SYSTEM CONVEYORS (* System Configuration *)
  (* Standard: 61499-1 *)
  (* Version 0.4, 2009-03-05, JHC, Holobloc Inc., Deleted Application. *)
  (* Version 0.3, 2003-12-05, JHC, Rockwell Automation, Renamed from NEWSYSTEM. *)
  (* Version 0.2, 2002-11-05, JHC, Rockwell Automation, Fixed missing (empty) FBD in Application. *)
  (* Version 0.1, 2002-01-17, JHC, Rockwell Automation, Minor cleanup *)
  (* Version 0.0, 2000-05-27, JHC, Rockwell Automation *)
  DEVICE VIEW : FRAME_DEVICE(BOUNDS := [500,30,520,500])
    RESOURCE VIEW_Resource : VIEW_PANEL(DIA := 50, SIZE := [10,10])
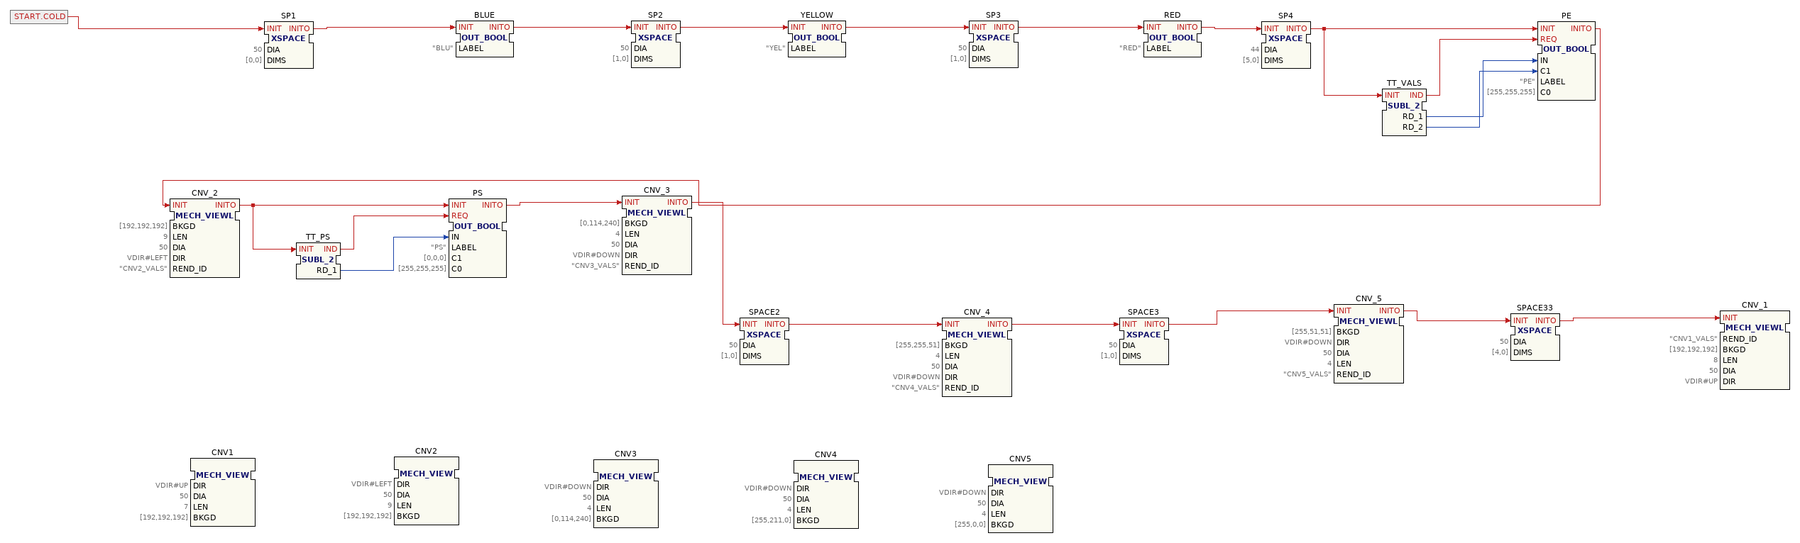
      FBS
        CNV1 : MECH_VIEW(DIR := VDIR#UP, DIA := 50, LEN := 7, BKGD := [192,192,192]);
        CNV2 : MECH_VIEW(DIR := VDIR#LEFT, DIA := 50, LEN := 9, BKGD := [192,192,192]);
        CNV3 : MECH_VIEW(DIR := VDIR#DOWN, DIA := 50, LEN := 4, BKGD := [0,114,240]);
        CNV4 : MECH_VIEW(DIR := VDIR#DOWN, DIA := 50, LEN := 4, BKGD := [255,211,0]);
        CNV5 : MECH_VIEW(DIR := VDIR#DOWN, DIA := 50, LEN := 4, BKGD := [255,0,0]);
        SPACE2 : XSPACE(DIA := 50, DIMS := [1,0]);
        SPACE3 : XSPACE(DIA := 50, DIMS := [1,0]);
        BLUE : OUT_BOOL(LABEL := "BLU");
        YELLOW : OUT_BOOL(LABEL := "YEL");
        RED : OUT_BOOL(LABEL := "RED");
        SP1 : XSPACE(DIA := 50, DIMS := [0,0]);
        SP2 : XSPACE(DIA := 50, DIMS := [1,0]);
        SP3 : XSPACE(DIA := 50, DIMS := [1,0]);
        SP4 : XSPACE(DIA := 44, DIMS := [5,0]);
        SPACE33 : XSPACE(DIA := 50, DIMS := [4,0]);
        PS : OUT_BOOL(LABEL := "PS", C1 := [0,0,0], C0 := [255,255,255]);
        PE : OUT_BOOL(LABEL := "PE", C0 := [255,255,255]);
        CNV_2 : MECH_VIEWL(BKGD := [192,192,192], LEN := 9, DIA := 50, DIR := VDIR#LEFT, REND_ID := "CNV2_VALS");
        CNV_3 : MECH_VIEWL(BKGD := [0,114,240], LEN := 4, DIA := 50, DIR := VDIR#DOWN, REND_ID := "CNV3_VALS");
        CNV_4 : MECH_VIEWL(BKGD := [255,255,51], LEN := 4, DIA := 50, DIR := VDIR#DOWN, REND_ID := "CNV4_VALS");
        CNV_5 : MECH_VIEWL(BKGD := [255,51,51], DIR := VDIR#DOWN, DIA := 50, LEN := 4, REND_ID := "CNV5_VALS");
        TT_VALS : SUBL_2;
        TT_PS : SUBL_2;
        CNV_1 : MECH_VIEWL(REND_ID := "CNV1_VALS", BKGD := [192,192,192], LEN := 8, DIA := 50, DIR := VDIR#UP);
      END_FBS
      EVENT_CONNECTIONS
        START.COLD TO SP1.INIT;
        SP1.INITO TO BLUE.INIT;
        BLUE.INITO TO SP2.INIT;
        SP2.INITO TO YELLOW.INIT;
        YELLOW.INITO TO SP3.INIT;
        SP3.INITO TO RED.INIT;
        RED.INITO TO SP4.INIT;
        SP4.INITO TO PE.INIT;
        PE.INITO TO CNV_2.INIT;
        CNV_2.INITO TO PS.INIT;
        PS.INITO TO CNV_3.INIT;
        CNV_3.INITO TO SPACE2.INIT;
        SPACE2.INITO TO CNV_4.INIT;
        CNV_4.INITO TO SPACE3.INIT;
        SPACE3.INITO TO CNV_5.INIT;
        CNV_5.INITO TO SPACE33.INIT;
        SP4.INITO TO TT_VALS.INIT;
        TT_VALS.IND TO PE.REQ;
        CNV_2.INITO TO TT_PS.INIT;
        TT_PS.IND TO PS.REQ;
        SPACE33.INITO TO CNV_1.INIT;
      END_CONNECTIONS
      DATA_CONNECTIONS
        TT_VALS.RD_1 TO PE.IN;
        TT_VALS.RD_2 TO PE.C1;
        TT_PS.RD_1 TO PS.IN;
      END_CONNECTIONS
    END_RESOURCE
  END_DEVICE
  DEVICE HMI : FRAME_DEVICE(BOUNDS := [1000,30,500,500])
    RESOURCE HMI_RESOURCE : VIEW_PANEL(DIA := 50, SIZE := [10,10])
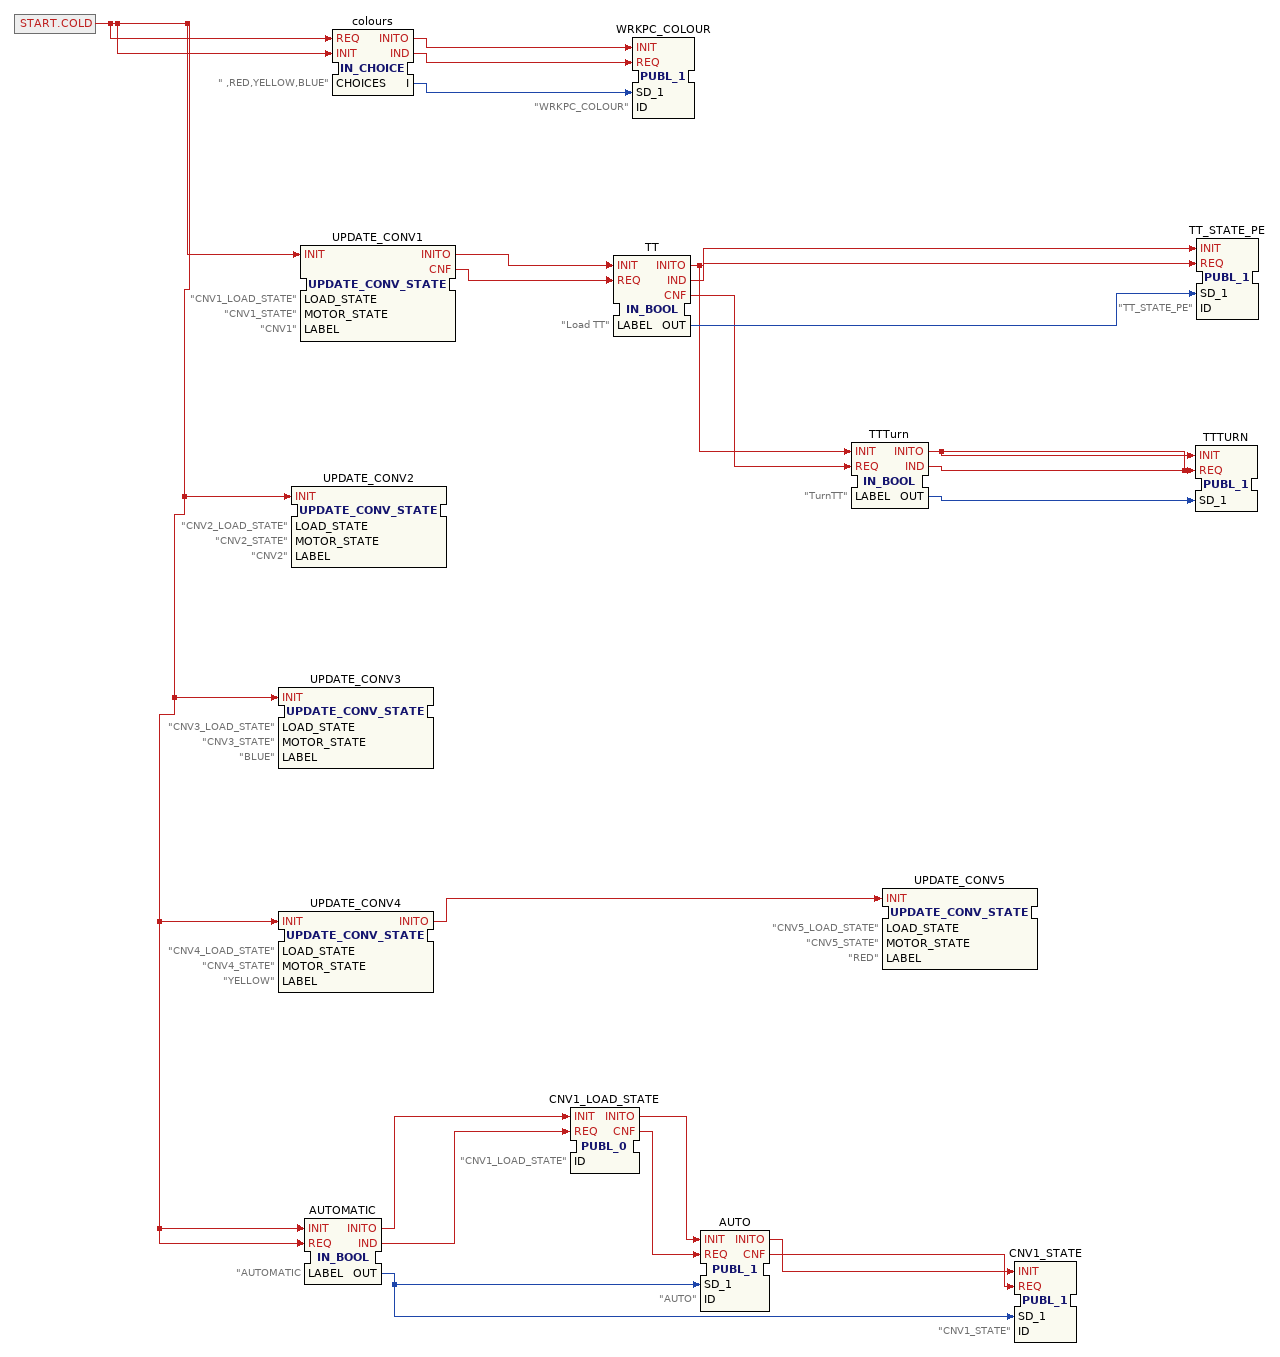
      FBS
        colours : IN_CHOICE(CHOICES := " ,RED,YELLOW,BLUE");
        WRKPC_COLOUR : PUBL_1(ID := "WRKPC_COLOUR");
        TT_STATE_PE : PUBL_1(ID := "TT_STATE_PE");
        TT : IN_BOOL(LABEL := "Load TT");
        TTTurn : IN_BOOL(LABEL := "TurnTT");
        TTTURN : PUBL_1;
        UPDATE_CONV1 : UPDATE_CONV_STATE(LOAD_STATE := "CNV1_LOAD_STATE", MOTOR_STATE := "CNV1_STATE", LABEL := "CNV1");
        UPDATE_CONV2 : UPDATE_CONV_STATE(LOAD_STATE := "CNV2_LOAD_STATE", MOTOR_STATE := "CNV2_STATE", LABEL := "CNV2");
        UPDATE_CONV3 : UPDATE_CONV_STATE(LOAD_STATE := "CNV3_LOAD_STATE", MOTOR_STATE := "CNV3_STATE", LABEL := "BLUE");
        UPDATE_CONV4 : UPDATE_CONV_STATE(LOAD_STATE := "CNV4_LOAD_STATE", MOTOR_STATE := "CNV4_STATE", LABEL := "YELLOW");
        UPDATE_CONV5 : UPDATE_CONV_STATE(LOAD_STATE := "CNV5_LOAD_STATE", MOTOR_STATE := "CNV5_STATE", LABEL := "RED");
        AUTOMATIC : IN_BOOL(LABEL := "AUTOMATIC);
        CNV1_STATE : PUBL_1(ID := "CNV1_STATE");
        CNV1_LOAD_STATE : PUBL_0(ID := "CNV1_LOAD_STATE");
        AUTO : PUBL_1(ID := "AUTO");
      END_FBS
      EVENT_CONNECTIONS
        START.COLD TO colours.REQ;
        START.COLD TO colours.INIT;
        colours.INITO TO WRKPC_COLOUR.INIT;
        colours.IND TO WRKPC_COLOUR.REQ;
        TT.INITO TO TT_STATE_PE.INIT;
        TT.IND TO TT_STATE_PE.REQ;
        TT.INITO TO TTTurn.INIT;
        TT.CNF TO TTTurn.REQ;
        TTTurn.INITO TO TTTURN.INIT;
        TTTurn.IND TO TTTURN.REQ;
        TTTurn.INITO TO TTTURN.REQ;
        START.COLD TO UPDATE_CONV1.INIT;
        UPDATE_CONV1.INITO TO TT.INIT;
        UPDATE_CONV1.CNF TO TT.REQ;
        START.COLD TO UPDATE_CONV2.INIT;
        START.COLD TO UPDATE_CONV3.INIT;
        START.COLD TO UPDATE_CONV4.INIT;
        UPDATE_CONV4.INITO TO UPDATE_CONV5.INIT;
        START.COLD TO AUTOMATIC.INIT;
        START.COLD TO AUTOMATIC.REQ;
        AUTOMATIC.INITO TO CNV1_LOAD_STATE.INIT;
        AUTOMATIC.IND TO CNV1_LOAD_STATE.REQ;
        CNV1_LOAD_STATE.INITO TO AUTO.INIT;
        CNV1_LOAD_STATE.CNF TO AUTO.REQ;
        AUTO.INITO TO CNV1_STATE.INIT;
        AUTO.CNF TO CNV1_STATE.REQ;
      END_CONNECTIONS
      DATA_CONNECTIONS
        colours.I TO WRKPC_COLOUR.SD_1;
        TT.OUT TO TT_STATE_PE.SD_1;
        TTTurn.OUT TO TTTURN.SD_1;
        AUTOMATIC.OUT TO CNV1_STATE.SD_1;
        AUTOMATIC.OUT TO AUTO.SD_1;
      END_CONNECTIONS
    END_RESOURCE
  END_DEVICE
  DEVICE MODEL : FRAME_DEVICE(BOUNDS := [500,570,500,500])
    RESOURCE CONV1_MODEL : VIEW_PANEL(DIA := 50, SIZE := [1,1])
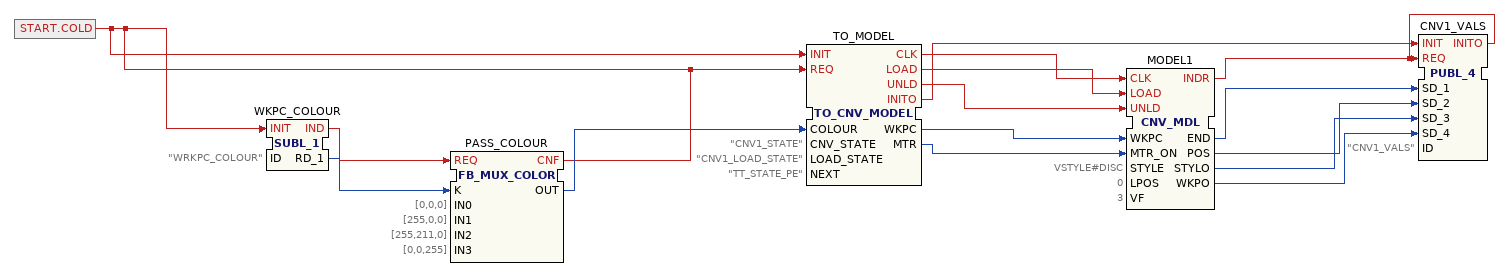
      FBS
        MODEL1 : CNV_MDL(STYLE := VSTYLE#DISC, LPOS := 0, VF := 3);
        TO_MODEL : TO_CNV_MODEL(CNV_STATE := "CNV1_STATE", LOAD_STATE := "CNV1_LOAD_STATE", NEXT := "TT_STATE_PE");
        CNV1_VALS : PUBL_4(ID := "CNV1_VALS");
        WKPC_COLOUR : SUBL_1(ID := "WRKPC_COLOUR");
        PASS_COLOUR : FB_MUX_COLOR(IN0 := [0,0,0], IN1 := [255,0,0], IN2 := [255,211,0], IN3 := [0,0,255]);
      END_FBS
      EVENT_CONNECTIONS
        START.COLD TO TO_MODEL.INIT;
        TO_MODEL.CLK TO MODEL1.CLK;
        START.COLD TO TO_MODEL.REQ;
        TO_MODEL.LOAD TO MODEL1.LOAD;
        TO_MODEL.UNLD TO MODEL1.UNLD;
        TO_MODEL.INITO TO CNV1_VALS.INIT;
        MODEL1.INDR TO CNV1_VALS.REQ;
        CNV1_VALS.INITO TO CNV1_VALS.REQ;
        START.COLD TO WKPC_COLOUR.INIT;
        WKPC_COLOUR.IND TO PASS_COLOUR.REQ;
        PASS_COLOUR.CNF TO TO_MODEL.REQ;
      END_CONNECTIONS
      DATA_CONNECTIONS
        TO_MODEL.WKPC TO MODEL1.WKPC;
        TO_MODEL.MTR TO MODEL1.MTR_ON;
        MODEL1.END TO CNV1_VALS.SD_1;
        MODEL1.POS TO CNV1_VALS.SD_2;
        MODEL1.STYLO TO CNV1_VALS.SD_3;
        MODEL1.WKPO TO CNV1_VALS.SD_4;
        WKPC_COLOUR.RD_1 TO PASS_COLOUR.K;
        PASS_COLOUR.OUT TO TO_MODEL.COLOUR;
      END_CONNECTIONS
    END_RESOURCE
    RESOURCE TT_MODEL : VIEW_PANEL(DIA := 50, SIZE := [1,1])
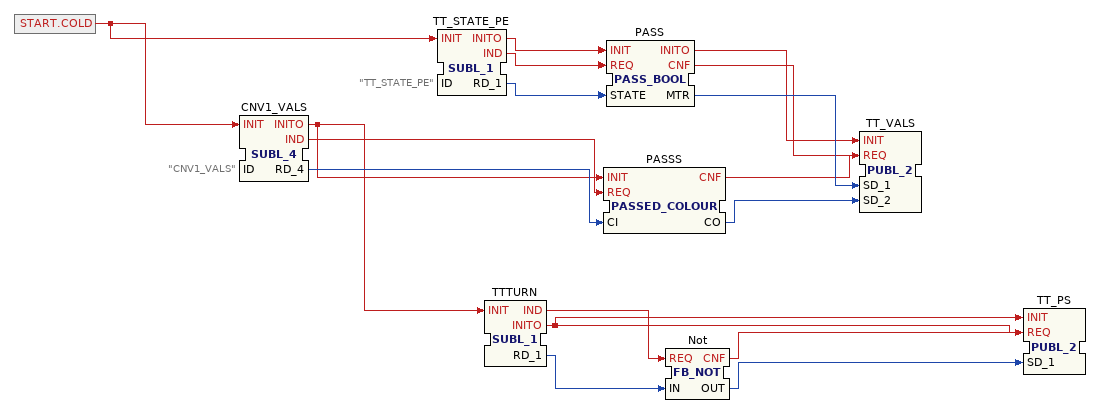
      FBS
        TT_STATE_PE : SUBL_1(ID := "TT_STATE_PE");
        TT_PS : PUBL_2;
        TTTURN : SUBL_1;
        Not : FB_NOT;
        CNV1_VALS : SUBL_4(ID := "CNV1_VALS");
        PASS : PASS_BOOL;
        PASSS : PASSED_COLOUR;
        TT_VALS : PUBL_2;
      END_FBS
      EVENT_CONNECTIONS
        START.COLD TO TT_STATE_PE.INIT;
        TTTURN.IND TO Not.REQ;
        TTTURN.INITO TO TT_PS.INIT;
        Not.CNF TO TT_PS.REQ;
        TTTURN.INITO TO TT_PS.REQ;
        START.COLD TO CNV1_VALS.INIT;
        CNV1_VALS.INITO TO TTTURN.INIT;
        TT_STATE_PE.INITO TO PASS.INIT;
        TT_STATE_PE.IND TO PASS.REQ;
        CNV1_VALS.INITO TO PASSS.INIT;
        CNV1_VALS.IND TO PASSS.REQ;
        PASS.INITO TO TT_VALS.INIT;
        PASS.CNF TO TT_VALS.REQ;
        PASSS.CNF TO TT_VALS.REQ;
      END_CONNECTIONS
      DATA_CONNECTIONS
        Not.OUT TO TT_PS.SD_1;
        TTTURN.RD_1 TO Not.IN;
        TT_STATE_PE.RD_1 TO PASS.STATE;
        CNV1_VALS.RD_4 TO PASSS.CI;
        PASS.MTR TO TT_VALS.SD_1;
        PASSS.CO TO TT_VALS.SD_2;
      END_CONNECTIONS
    END_RESOURCE
    RESOURCE CONV2_MODEL : VIEW_PANEL(DIA := 50, SIZE := [1,1])
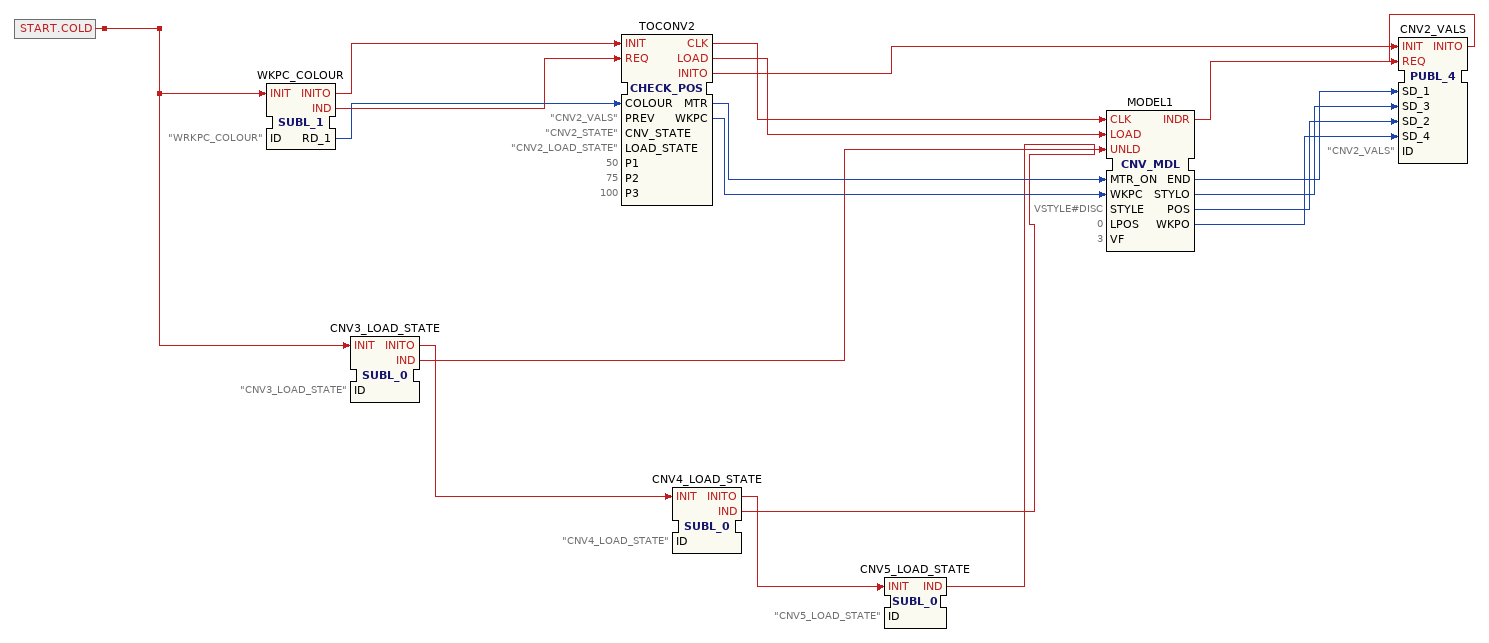
      FBS
        MODEL1 : CNV_MDL(STYLE := VSTYLE#DISC, LPOS := 0, VF := 3);
        TOCONV2 : CHECK_POS(PREV := "CNV2_VALS", CNV_STATE := "CNV2_STATE", LOAD_STATE := "CNV2_LOAD_STATE", P1 := 50, P2 := 75, P3 := 100);
        CNV3_LOAD_STATE : SUBL_0(ID := "CNV3_LOAD_STATE");
        CNV4_LOAD_STATE : SUBL_0(ID := "CNV4_LOAD_STATE");
        CNV5_LOAD_STATE : SUBL_0(ID := "CNV5_LOAD_STATE");
        CNV2_VALS : PUBL_4(ID := "CNV2_VALS");
        WKPC_COLOUR : SUBL_1(ID := "WRKPC_COLOUR");
      END_FBS
      EVENT_CONNECTIONS
        TOCONV2.CLK TO MODEL1.CLK;
        TOCONV2.LOAD TO MODEL1.LOAD;
        CNV3_LOAD_STATE.INITO TO CNV4_LOAD_STATE.INIT;
        CNV4_LOAD_STATE.INITO TO CNV5_LOAD_STATE.INIT;
        TOCONV2.INITO TO CNV2_VALS.INIT;
        MODEL1.INDR TO CNV2_VALS.REQ;
        CNV2_VALS.INITO TO CNV2_VALS.REQ;
        START.COLD TO WKPC_COLOUR.INIT;
        WKPC_COLOUR.INITO TO TOCONV2.INIT;
        WKPC_COLOUR.IND TO TOCONV2.REQ;
        START.COLD TO CNV3_LOAD_STATE.INIT;
        CNV3_LOAD_STATE.IND TO MODEL1.UNLD;
        CNV4_LOAD_STATE.IND TO MODEL1.UNLD;
        CNV5_LOAD_STATE.IND TO MODEL1.UNLD;
      END_CONNECTIONS
      DATA_CONNECTIONS
        TOCONV2.MTR TO MODEL1.MTR_ON;
        TOCONV2.WKPC TO MODEL1.WKPC;
        MODEL1.END TO CNV2_VALS.SD_1;
        MODEL1.STYLO TO CNV2_VALS.SD_3;
        MODEL1.POS TO CNV2_VALS.SD_2;
        MODEL1.WKPO TO CNV2_VALS.SD_4;
        WKPC_COLOUR.RD_1 TO TOCONV2.COLOUR;
      END_CONNECTIONS
    END_RESOURCE
    RESOURCE CONV3_MODEL : VIEW_PANEL(DIA := 50, SIZE := [1,1])
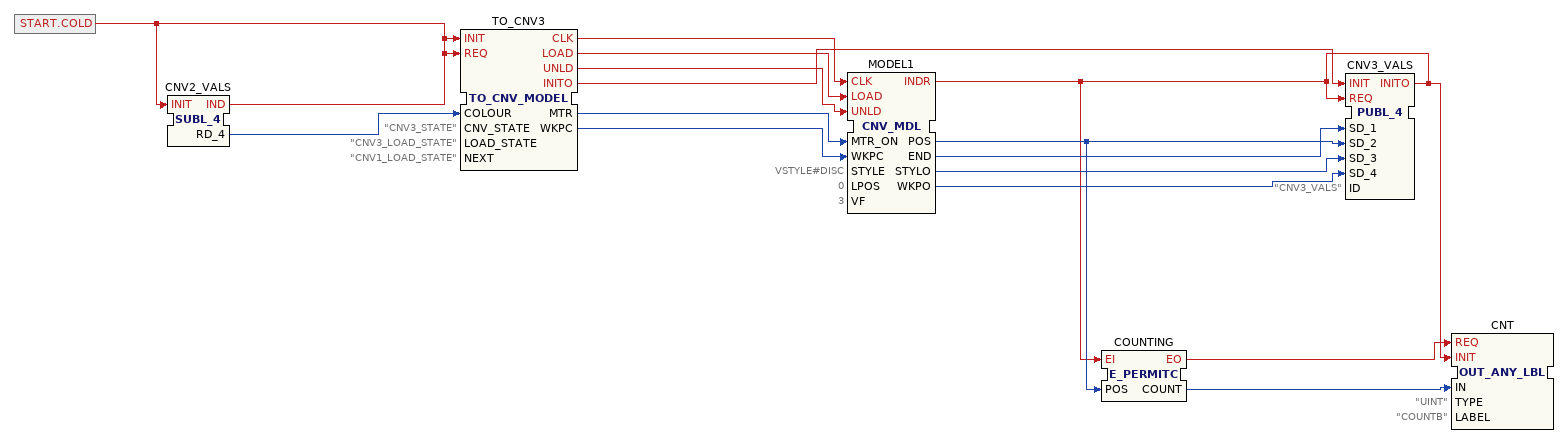
      FBS
        MODEL1 : CNV_MDL(STYLE := VSTYLE#DISC, LPOS := 0, VF := 3);
        TO_CNV3 : TO_CNV_MODEL(CNV_STATE := "CNV3_STATE", LOAD_STATE := "CNV3_LOAD_STATE", NEXT := "CNV1_LOAD_STATE");
        COUNTING : E_PERMITC;
        CNT : OUT_ANY_LBL(TYPE := "UINT", LABEL := "COUNTB");
        CNV3_VALS : PUBL_4(ID := "CNV3_VALS");
        CNV2_VALS : SUBL_4;
      END_FBS
      EVENT_CONNECTIONS
        START.COLD TO TO_CNV3.INIT;
        START.COLD TO TO_CNV3.REQ;
        TO_CNV3.CLK TO MODEL1.CLK;
        TO_CNV3.LOAD TO MODEL1.LOAD;
        TO_CNV3.UNLD TO MODEL1.UNLD;
        MODEL1.INDR TO COUNTING.EI;
        COUNTING.EO TO CNT.REQ;
        TO_CNV3.INITO TO CNV3_VALS.INIT;
        MODEL1.INDR TO CNV3_VALS.REQ;
        CNV3_VALS.INITO TO CNV3_VALS.REQ;
        CNV3_VALS.INITO TO CNT.INIT;
        START.COLD TO CNV2_VALS.INIT;
        CNV2_VALS.IND TO TO_CNV3.REQ;
      END_CONNECTIONS
      DATA_CONNECTIONS
        TO_CNV3.MTR TO MODEL1.MTR_ON;
        TO_CNV3.WKPC TO MODEL1.WKPC;
        MODEL1.POS TO COUNTING.POS;
        COUNTING.COUNT TO CNT.IN;
        MODEL1.END TO CNV3_VALS.SD_1;
        MODEL1.POS TO CNV3_VALS.SD_2;
        MODEL1.STYLO TO CNV3_VALS.SD_3;
        MODEL1.WKPO TO CNV3_VALS.SD_4;
        CNV2_VALS.RD_4 TO TO_CNV3.COLOUR;
      END_CONNECTIONS
    END_RESOURCE
    RESOURCE CONV4_MODEL : VIEW_PANEL(DIA := 50, SIZE := [1,1])
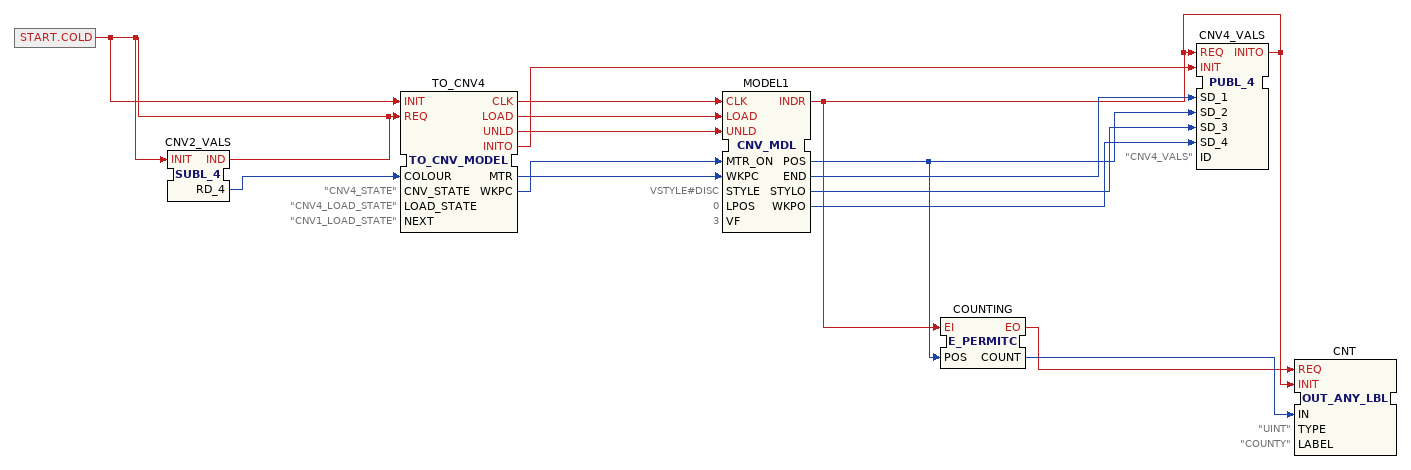
      FBS
        MODEL1 : CNV_MDL(STYLE := VSTYLE#DISC, LPOS := 0, VF := 3);
        TO_CNV4 : TO_CNV_MODEL(CNV_STATE := "CNV4_STATE", LOAD_STATE := "CNV4_LOAD_STATE", NEXT := "CNV1_LOAD_STATE");
        COUNTING : E_PERMITC;
        CNT : OUT_ANY_LBL(TYPE := "UINT", LABEL := "COUNTY");
        CNV4_VALS : PUBL_4(ID := "CNV4_VALS");
        CNV2_VALS : SUBL_4;
      END_FBS
      EVENT_CONNECTIONS
        START.COLD TO TO_CNV4.INIT;
        TO_CNV4.CLK TO MODEL1.CLK;
        TO_CNV4.LOAD TO MODEL1.LOAD;
        TO_CNV4.UNLD TO MODEL1.UNLD;
        START.COLD TO TO_CNV4.REQ;
        MODEL1.INDR TO COUNTING.EI;
        COUNTING.EO TO CNT.REQ;
        CNV4_VALS.INITO TO CNV4_VALS.REQ;
        TO_CNV4.INITO TO CNV4_VALS.INIT;
        MODEL1.INDR TO CNV4_VALS.REQ;
        CNV4_VALS.INITO TO CNT.INIT;
        START.COLD TO CNV2_VALS.INIT;
        CNV2_VALS.IND TO TO_CNV4.REQ;
      END_CONNECTIONS
      DATA_CONNECTIONS
        TO_CNV4.MTR TO MODEL1.MTR_ON;
        TO_CNV4.WKPC TO MODEL1.WKPC;
        MODEL1.POS TO COUNTING.POS;
        COUNTING.COUNT TO CNT.IN;
        MODEL1.END TO CNV4_VALS.SD_1;
        MODEL1.POS TO CNV4_VALS.SD_2;
        MODEL1.STYLO TO CNV4_VALS.SD_3;
        MODEL1.WKPO TO CNV4_VALS.SD_4;
        CNV2_VALS.RD_4 TO TO_CNV4.COLOUR;
      END_CONNECTIONS
    END_RESOURCE
    RESOURCE CONV5_MODEL : VIEW_PANEL(DIA := 50, SIZE := [1,1])
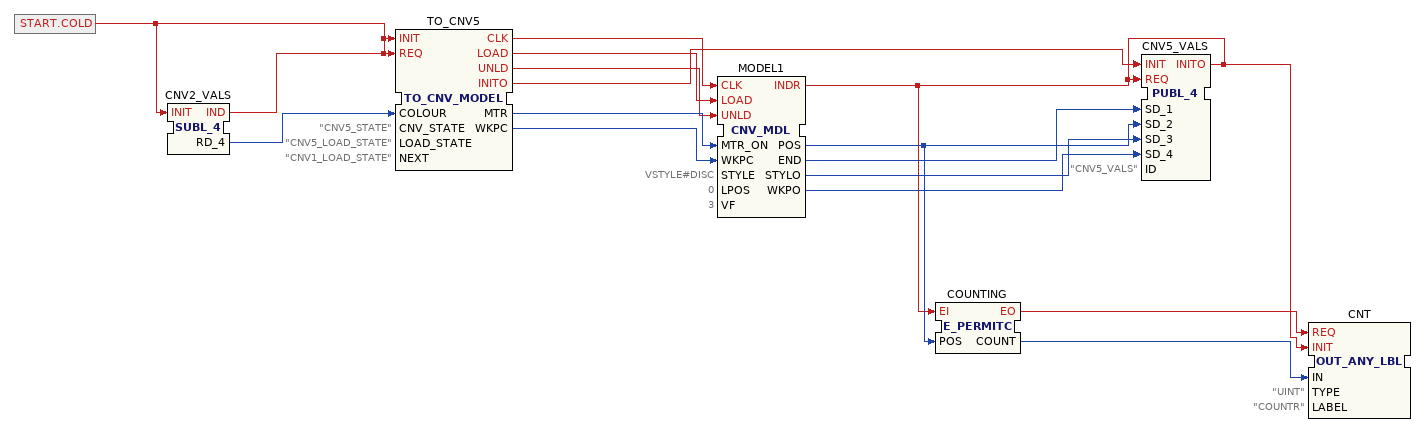
      FBS
        MODEL1 : CNV_MDL(STYLE := VSTYLE#DISC, LPOS := 0, VF := 3);
        TO_CNV5 : TO_CNV_MODEL(CNV_STATE := "CNV5_STATE", LOAD_STATE := "CNV5_LOAD_STATE", NEXT := "CNV1_LOAD_STATE");
        COUNTING : E_PERMITC;
        CNT : OUT_ANY_LBL(TYPE := "UINT", LABEL := "COUNTR");
        CNV5_VALS : PUBL_4(ID := "CNV5_VALS");
        CNV2_VALS : SUBL_4;
      END_FBS
      EVENT_CONNECTIONS
        START.COLD TO TO_CNV5.INIT;
        START.COLD TO TO_CNV5.REQ;
        TO_CNV5.CLK TO MODEL1.CLK;
        TO_CNV5.LOAD TO MODEL1.LOAD;
        TO_CNV5.UNLD TO MODEL1.UNLD;
        MODEL1.INDR TO COUNTING.EI;
        COUNTING.EO TO CNT.REQ;
        TO_CNV5.INITO TO CNV5_VALS.INIT;
        MODEL1.INDR TO CNV5_VALS.REQ;
        CNV5_VALS.INITO TO CNV5_VALS.REQ;
        CNV5_VALS.INITO TO CNT.INIT;
        START.COLD TO CNV2_VALS.INIT;
        CNV2_VALS.IND TO TO_CNV5.REQ;
      END_CONNECTIONS
      DATA_CONNECTIONS
        TO_CNV5.MTR TO MODEL1.MTR_ON;
        TO_CNV5.WKPC TO MODEL1.WKPC;
        MODEL1.POS TO COUNTING.POS;
        COUNTING.COUNT TO CNT.IN;
        MODEL1.END TO CNV5_VALS.SD_1;
        MODEL1.POS TO CNV5_VALS.SD_2;
        MODEL1.STYLO TO CNV5_VALS.SD_3;
        MODEL1.WKPO TO CNV5_VALS.SD_4;
        CNV2_VALS.RD_4 TO TO_CNV5.COLOUR;
      END_CONNECTIONS
    END_RESOURCE
  END_DEVICE
  DEVICE CONTROL : FRAME_DEVICE(BOUNDS := [1000,570,500,500])
    RESOURCE CONV1_CTRL : VIEW_PANEL(DIA := 50, SIZE := [1,1])
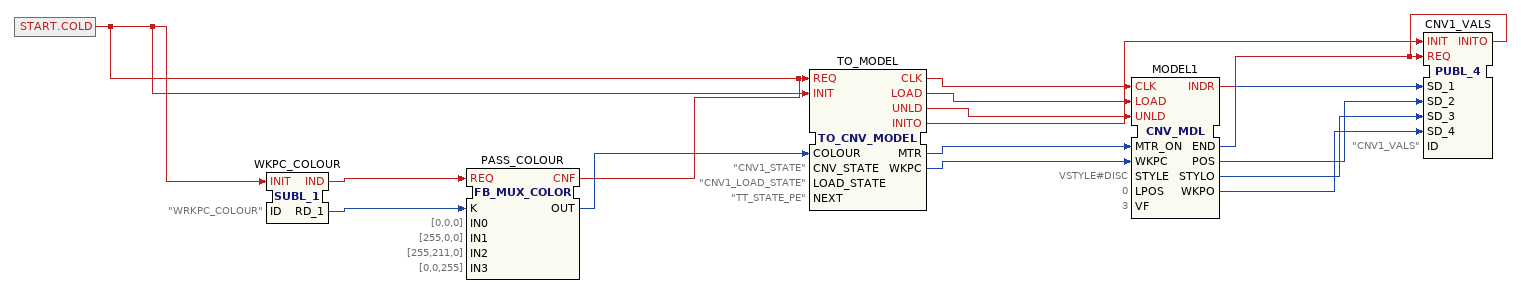
      FBS
        MODEL1 : CNV_MDL(STYLE := VSTYLE#DISC, LPOS := 0, VF := 3);
        TO_MODEL : TO_CNV_MODEL(CNV_STATE := "CNV1_STATE", LOAD_STATE := "CNV1_LOAD_STATE", NEXT := "TT_STATE_PE");
        CNV1_VALS : PUBL_4(ID := "CNV1_VALS");
        WKPC_COLOUR : SUBL_1(ID := "WRKPC_COLOUR");
        PASS_COLOUR : FB_MUX_COLOR(IN0 := [0,0,0], IN1 := [255,0,0], IN2 := [255,211,0], IN3 := [0,0,255]);
      END_FBS
      EVENT_CONNECTIONS
        START.COLD TO TO_MODEL.REQ;
        TO_MODEL.CLK TO MODEL1.CLK;
        TO_MODEL.LOAD TO MODEL1.LOAD;
        TO_MODEL.UNLD TO MODEL1.UNLD;
        TO_MODEL.INITO TO CNV1_VALS.INIT;
        MODEL1.INDR TO CNV1_VALS.REQ;
        START.COLD TO TO_MODEL.INIT;
        CNV1_VALS.INITO TO CNV1_VALS.REQ;
        START.COLD TO WKPC_COLOUR.INIT;
        WKPC_COLOUR.IND TO PASS_COLOUR.REQ;
        PASS_COLOUR.CNF TO TO_MODEL.REQ;
      END_CONNECTIONS
      DATA_CONNECTIONS
        TO_MODEL.MTR TO MODEL1.MTR_ON;
        TO_MODEL.WKPC TO MODEL1.WKPC;
        MODEL1.END TO CNV1_VALS.SD_1;
        MODEL1.POS TO CNV1_VALS.SD_2;
        MODEL1.STYLO TO CNV1_VALS.SD_3;
        MODEL1.WKPO TO CNV1_VALS.SD_4;
        WKPC_COLOUR.RD_1 TO PASS_COLOUR.K;
        PASS_COLOUR.OUT TO TO_MODEL.COLOUR;
      END_CONNECTIONS
    END_RESOURCE
    RESOURCE TT_CTRL : VIEW_PANEL(DIA := 50, SIZE := [1,1])
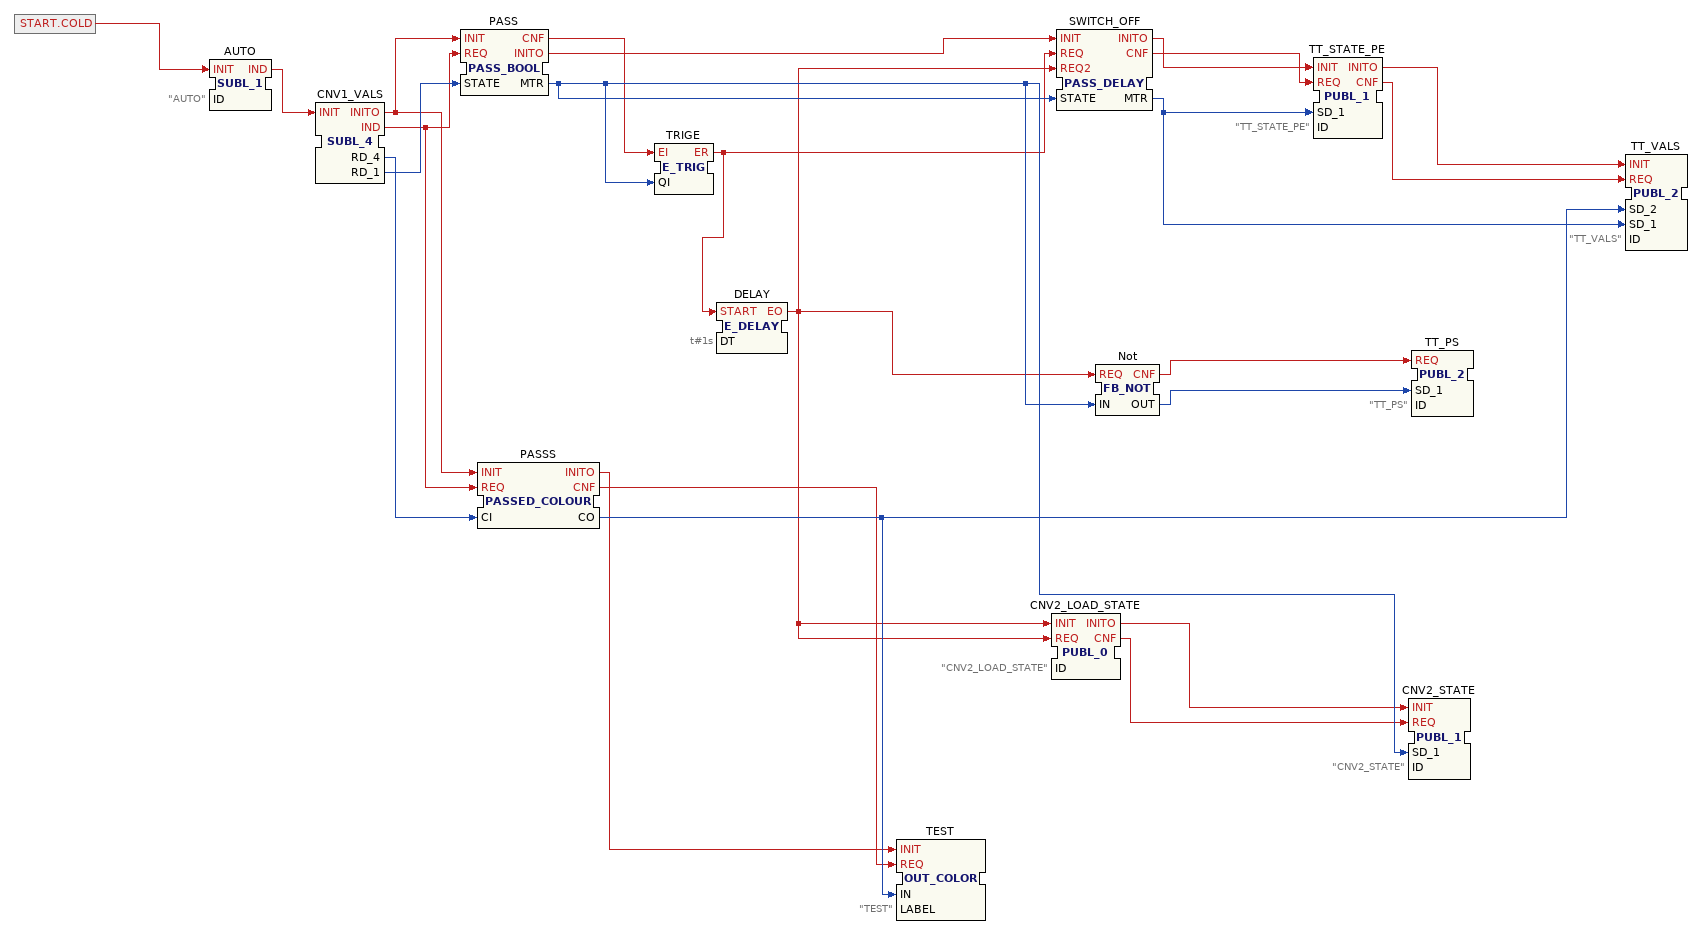
      FBS
        TT_PS : PUBL_2(ID := "TT_PS");
        DELAY : E_DELAY(DT := t#1s);
        Not : FB_NOT;
        CNV2_LOAD_STATE : PUBL_0(ID := "CNV2_LOAD_STATE");
        CNV2_STATE : PUBL_1(ID := "CNV2_STATE");
        PASS : PASS_BOOL;
        PASSS : PASSED_COLOUR;
        CNV1_VALS : SUBL_4;
        TT_STATE_PE : PUBL_1(ID := "TT_STATE_PE");
        AUTO : SUBL_1(ID := "AUTO");
        TT_VALS : PUBL_2(ID := "TT_VALS");
        TRIGE : E_TRIG;
        SWITCH_OFF : PASS_DELAY;
        TEST : OUT_COLOR(LABEL := "TEST");
      END_FBS
      EVENT_CONNECTIONS
        Not.CNF TO TT_PS.REQ;
        CNV2_LOAD_STATE.INITO TO CNV2_STATE.INIT;
        CNV1_VALS.INITO TO PASS.INIT;
        CNV1_VALS.IND TO PASS.REQ;
        CNV1_VALS.INITO TO PASSS.INIT;
        CNV1_VALS.IND TO PASSS.REQ;
        DELAY.EO TO Not.REQ;
        START.COLD TO AUTO.INIT;
        AUTO.IND TO CNV1_VALS.INIT;
        CNV2_LOAD_STATE.CNF TO CNV2_STATE.REQ;
        PASS.CNF TO TRIGE.EI;
        TRIGE.ER TO DELAY.START;
        TT_STATE_PE.INITO TO TT_VALS.INIT;
        TT_STATE_PE.CNF TO TT_VALS.REQ;
        PASS.INITO TO SWITCH_OFF.INIT;
        TRIGE.ER TO SWITCH_OFF.REQ;
        DELAY.EO TO SWITCH_OFF.REQ2;
        SWITCH_OFF.INITO TO TT_STATE_PE.INIT;
        SWITCH_OFF.CNF TO TT_STATE_PE.REQ;
        DELAY.EO TO CNV2_LOAD_STATE.INIT;
        DELAY.EO TO CNV2_LOAD_STATE.REQ;
        PASSS.INITO TO TEST.INIT;
        PASSS.CNF TO TEST.REQ;
      END_CONNECTIONS
      DATA_CONNECTIONS
        Not.OUT TO TT_PS.SD_1;
        CNV1_VALS.RD_4 TO PASSS.CI;
        PASS.MTR TO Not.IN;
        CNV1_VALS.RD_1 TO PASS.STATE;
        PASSS.CO TO TT_VALS.SD_2;
        PASS.MTR TO CNV2_STATE.SD_1;
        PASS.MTR TO TRIGE.QI;
        SWITCH_OFF.MTR TO TT_STATE_PE.SD_1;
        PASS.MTR TO SWITCH_OFF.STATE;
        SWITCH_OFF.MTR TO TT_VALS.SD_1;
        PASSS.CO TO TEST.IN;
      END_CONNECTIONS
    END_RESOURCE
    RESOURCE CONV2_CTRL : VIEW_PANEL(DIA := 50, SIZE := [1,1])
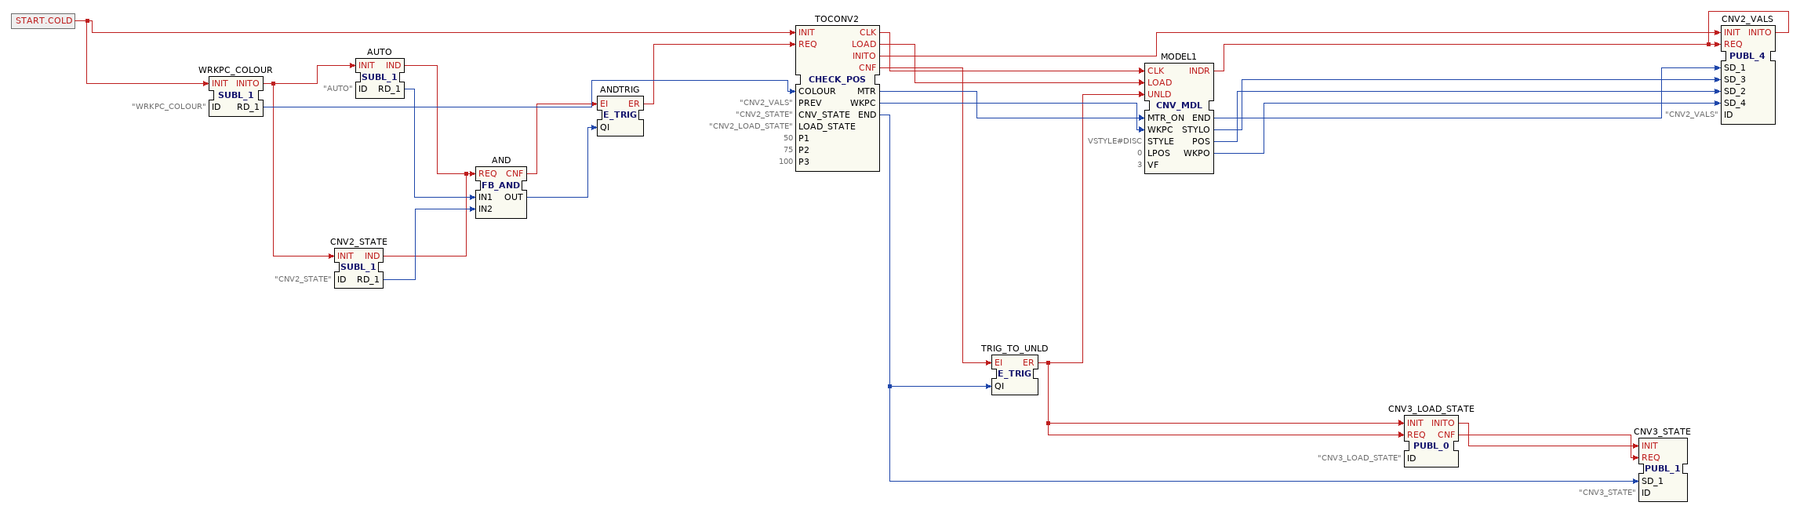
      FBS
        WRKPC_COLOUR : SUBL_1(ID := "WRKPC_COLOUR");
        MODEL1 : CNV_MDL(STYLE := VSTYLE#DISC, LPOS := 0, VF := 3);
        TOCONV2 : CHECK_POS(PREV := "CNV2_VALS", CNV_STATE := "CNV2_STATE", LOAD_STATE := "CNV2_LOAD_STATE", P1 := 50, P2 := 75, P3 := 100);
        CNV2_VALS : PUBL_4(ID := "CNV2_VALS");
        AUTO : SUBL_1(ID := "AUTO");
        CNV2_STATE : SUBL_1(ID := "CNV2_STATE");
        AND : FB_AND;
        ANDTRIG : E_TRIG;
        TRIG_TO_UNLD : E_TRIG;
        CNV3_LOAD_STATE : PUBL_0(ID := "CNV3_LOAD_STATE");
        CNV3_STATE : PUBL_1(ID := "CNV3_STATE");
      END_FBS
      EVENT_CONNECTIONS
        START.COLD TO WRKPC_COLOUR.INIT;
        START.COLD TO TOCONV2.INIT;
        TOCONV2.CLK TO MODEL1.CLK;
        TOCONV2.LOAD TO MODEL1.LOAD;
        TOCONV2.INITO TO CNV2_VALS.INIT;
        MODEL1.INDR TO CNV2_VALS.REQ;
        CNV2_VALS.INITO TO CNV2_VALS.REQ;
        WRKPC_COLOUR.INITO TO AUTO.INIT;
        WRKPC_COLOUR.INITO TO CNV2_STATE.INIT;
        AUTO.IND TO AND.REQ;
        CNV2_STATE.IND TO AND.REQ;
        AND.CNF TO ANDTRIG.EI;
        ANDTRIG.ER TO TOCONV2.REQ;
        TOCONV2.CNF TO TRIG_TO_UNLD.EI;
        TRIG_TO_UNLD.ER TO MODEL1.UNLD;
        TRIG_TO_UNLD.ER TO CNV3_LOAD_STATE.INIT;
        TRIG_TO_UNLD.ER TO CNV3_LOAD_STATE.REQ;
        CNV3_LOAD_STATE.INITO TO CNV3_STATE.INIT;
        CNV3_LOAD_STATE.CNF TO CNV3_STATE.REQ;
      END_CONNECTIONS
      DATA_CONNECTIONS
        TOCONV2.MTR TO MODEL1.MTR_ON;
        TOCONV2.WKPC TO MODEL1.WKPC;
        MODEL1.END TO CNV2_VALS.SD_1;
        MODEL1.STYLO TO CNV2_VALS.SD_3;
        MODEL1.POS TO CNV2_VALS.SD_2;
        MODEL1.WKPO TO CNV2_VALS.SD_4;
        WRKPC_COLOUR.RD_1 TO TOCONV2.COLOUR;
        AUTO.RD_1 TO AND.IN1;
        CNV2_STATE.RD_1 TO AND.IN2;
        AND.OUT TO ANDTRIG.QI;
        TOCONV2.END TO TRIG_TO_UNLD.QI;
        TOCONV2.END TO CNV3_STATE.SD_1;
      END_CONNECTIONS
    END_RESOURCE
    RESOURCE CONV3_CTRL : VIEW_PANEL(DIA := 50, SIZE := [1,1])
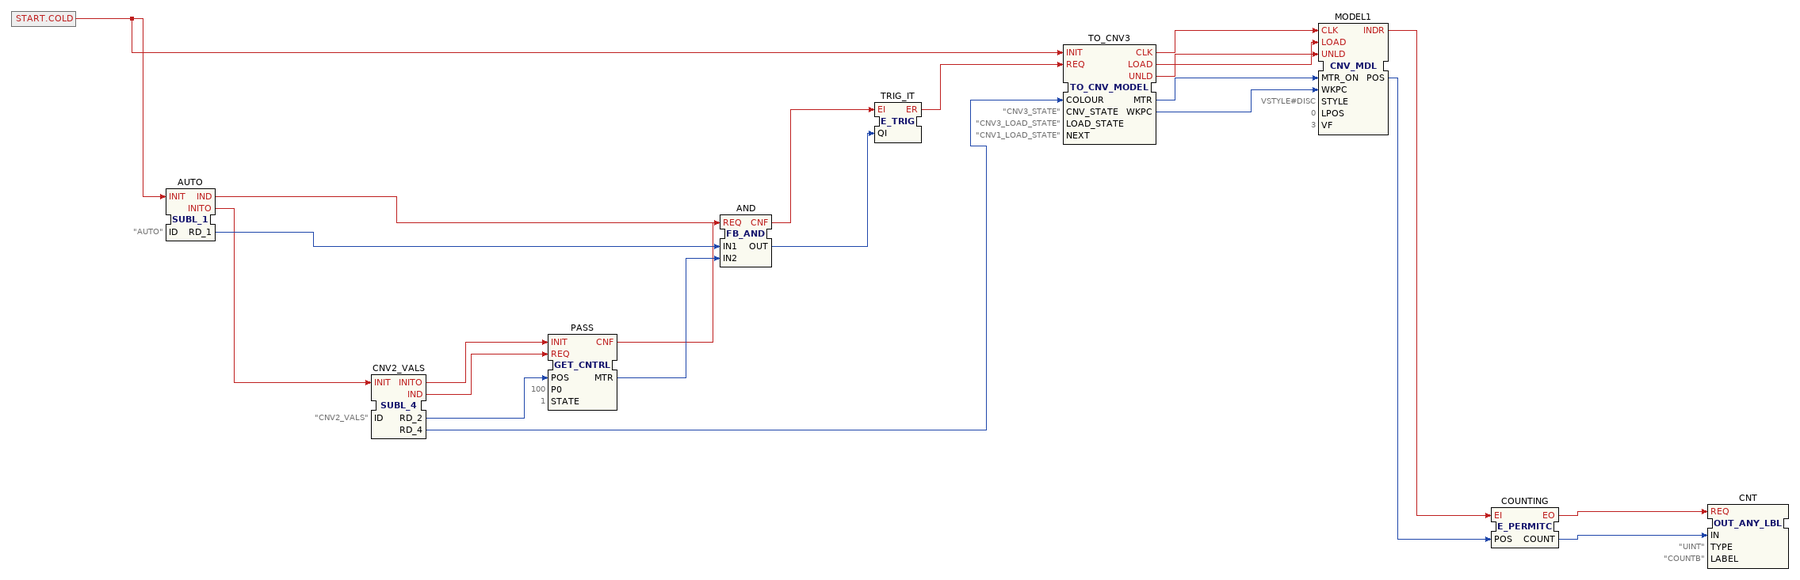
      FBS
        MODEL1 : CNV_MDL(STYLE := VSTYLE#DISC, LPOS := 0, VF := 3);
        TO_CNV3 : TO_CNV_MODEL(CNV_STATE := "CNV3_STATE", LOAD_STATE := "CNV3_LOAD_STATE", NEXT := "CNV1_LOAD_STATE");
        COUNTING : E_PERMITC;
        CNT : OUT_ANY_LBL(TYPE := "UINT", LABEL := "COUNTB");
        CNV2_VALS : SUBL_4(ID := "CNV2_VALS");
        PASS : GET_CNTRL(P0 := 100, STATE := 1);
        AUTO : SUBL_1(ID := "AUTO");
        AND : FB_AND;
        TRIG_IT : E_TRIG;
      END_FBS
      EVENT_CONNECTIONS
        TO_CNV3.CLK TO MODEL1.CLK;
        TO_CNV3.LOAD TO MODEL1.LOAD;
        TO_CNV3.UNLD TO MODEL1.UNLD;
        MODEL1.INDR TO COUNTING.EI;
        COUNTING.EO TO CNT.REQ;
        CNV2_VALS.INITO TO PASS.INIT;
        CNV2_VALS.IND TO PASS.REQ;
        AUTO.IND TO AND.REQ;
        START.COLD TO TO_CNV3.INIT;
        AUTO.INITO TO CNV2_VALS.INIT;
        START.COLD TO AUTO.INIT;
        AND.CNF TO TRIG_IT.EI;
        PASS.CNF TO AND.REQ;
        TRIG_IT.ER TO TO_CNV3.REQ;
      END_CONNECTIONS
      DATA_CONNECTIONS
        TO_CNV3.MTR TO MODEL1.MTR_ON;
        TO_CNV3.WKPC TO MODEL1.WKPC;
        MODEL1.POS TO COUNTING.POS;
        COUNTING.COUNT TO CNT.IN;
        CNV2_VALS.RD_2 TO PASS.POS;
        AUTO.RD_1 TO AND.IN1;
        CNV2_VALS.RD_4 TO TO_CNV3.COLOUR;
        AND.OUT TO TRIG_IT.QI;
        PASS.MTR TO AND.IN2;
      END_CONNECTIONS
    END_RESOURCE
    RESOURCE CONV4_CTRL : VIEW_PANEL(DIA := 50, SIZE := [1,1])
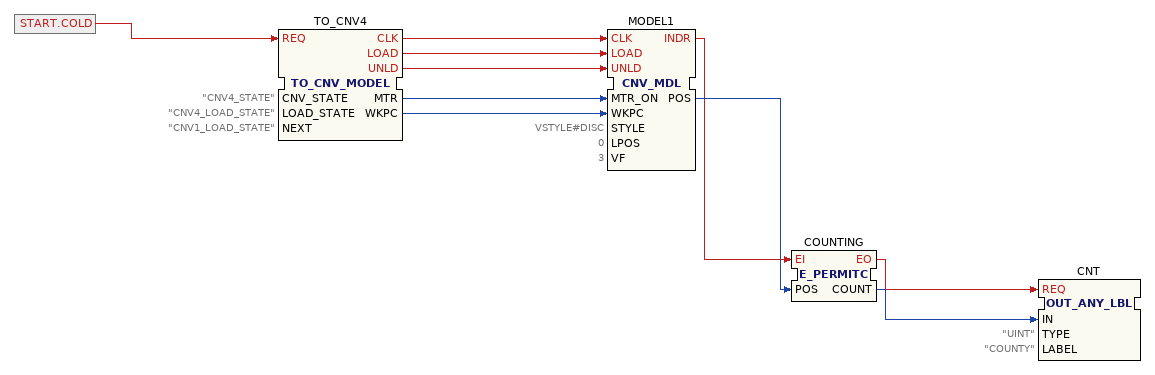
      FBS
        MODEL1 : CNV_MDL(STYLE := VSTYLE#DISC, LPOS := 0, VF := 3);
        TO_CNV4 : TO_CNV_MODEL(CNV_STATE := "CNV4_STATE", LOAD_STATE := "CNV4_LOAD_STATE", NEXT := "CNV1_LOAD_STATE");
        COUNTING : E_PERMITC;
        CNT : OUT_ANY_LBL(TYPE := "UINT", LABEL := "COUNTY");
      END_FBS
      EVENT_CONNECTIONS
        TO_CNV4.CLK TO MODEL1.CLK;
        TO_CNV4.LOAD TO MODEL1.LOAD;
        TO_CNV4.UNLD TO MODEL1.UNLD;
        START.COLD TO TO_CNV4.REQ;
        MODEL1.INDR TO COUNTING.EI;
        COUNTING.EO TO CNT.REQ;
      END_CONNECTIONS
      DATA_CONNECTIONS
        TO_CNV4.MTR TO MODEL1.MTR_ON;
        TO_CNV4.WKPC TO MODEL1.WKPC;
        MODEL1.POS TO COUNTING.POS;
        COUNTING.COUNT TO CNT.IN;
      END_CONNECTIONS
    END_RESOURCE
    RESOURCE CONV5_CTRL : VIEW_PANEL(DIA := 50, SIZE := [1,1])
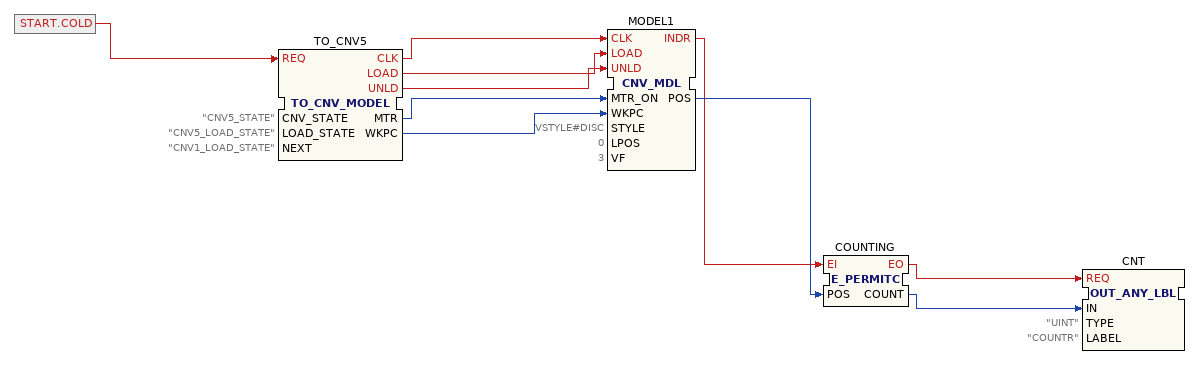
      FBS
        MODEL1 : CNV_MDL(STYLE := VSTYLE#DISC, LPOS := 0, VF := 3);
        TO_CNV5 : TO_CNV_MODEL(CNV_STATE := "CNV5_STATE", LOAD_STATE := "CNV5_LOAD_STATE", NEXT := "CNV1_LOAD_STATE");
        COUNTING : E_PERMITC;
        CNT : OUT_ANY_LBL(TYPE := "UINT", LABEL := "COUNTR");
      END_FBS
      EVENT_CONNECTIONS
        START.COLD TO TO_CNV5.REQ;
        TO_CNV5.CLK TO MODEL1.CLK;
        TO_CNV5.LOAD TO MODEL1.LOAD;
        TO_CNV5.UNLD TO MODEL1.UNLD;
        MODEL1.INDR TO COUNTING.EI;
        COUNTING.EO TO CNT.REQ;
      END_CONNECTIONS
      DATA_CONNECTIONS
        TO_CNV5.MTR TO MODEL1.MTR_ON;
        TO_CNV5.WKPC TO MODEL1.WKPC;
        MODEL1.POS TO COUNTING.POS;
        COUNTING.COUNT TO CNT.IN;
      END_CONNECTIONS
    END_RESOURCE
  END_DEVICE
END_SYSTEM
